(* PLC project Unnamed, Unknown Unnamed 1 *)
(* stored: creationDateTime 2026-02-04T10:46:58, modificationDateTime 2026-02-04T10:46:58 *)

PROGRAM main
  VAR
    Input_Switch AT %IX0.0 : BOOL;
    Output_Indicator AT %QX0.0 : BOOL;
  END_VAR

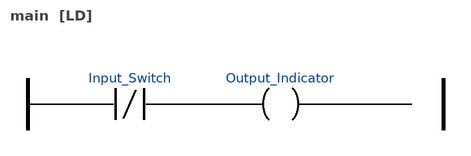
(* LD diagram, written out as Structured Text *)
Output_Indicator := NOT Input_Switch;
END_PROGRAM

CONFIGURATION Config0
  RESOURCE Res0 ON PLC
    TASK task0(INTERVAL := T#20ms, PRIORITY := 1);
    PROGRAM instance0 WITH task0 : main;
  END_RESOURCE
END_CONFIGURATION
